{attribute 'GeneratedUsingTerminal: EL5102-0000-0016'}
{attribute addProperty BoxType "EL5102-0000-0016"}
{attribute addProperty Id "ENC_Status_Channel_1AT %I*ENC_Status_Channel_10A67E5232ENC_Status_Channel_2AT %I*ENC_Status_Channel_10A67E5232ENC_Control_Channel_1AT %Q*ENC_Control_Channel_4C8A739514ENC_Control_Channel_2AT %Q*ENC_Control_Channel_4C8A739514WcStateAT %I*WcState_9091E0EB2InfoDataAT %I*InfoData_32EB74EA10"}
{attribute addProperty CRC "2140550683"}
{attribute addProperty Size "104"}
TYPE EL5102_7F96361B EXTENDS EtcSlaveTerminalBase_947E5A46 :
STRUCT
	{attribute addProperty Name "ENC_Status_Channel_1"}
	ENC_Status_Channel_1 : ENC_Status_Channel_10A67E52;
	{attribute addProperty Name "ENC_Status_Channel_2"}
	ENC_Status_Channel_2 : ENC_Status_Channel_10A67E52;
	{attribute addProperty Name "ENC_Control_Channel_1"}
	ENC_Control_Channel_1 : ENC_Control_Channel_4C8A7395;
	{attribute addProperty Name "ENC_Control_Channel_2"}
	ENC_Control_Channel_2 : ENC_Control_Channel_4C8A7395;
	{attribute addProperty Name "WcState"}
	WcState : WcState_9091E0EB;
	{attribute addProperty Name "InfoData"}
	InfoData : InfoData_32EB74EA;
END_STRUCT
END_TYPE

(* stored: Version 1.2.0.0, ProductVersion 3.1.4024.9
   DUT EL5102_7F96361B: Id {c6149bf6-64a4-4998-900a-79daf42393d4} *)
